FUNCTION_BLOCK FB_SetAxisMotion
VAR_IN_OUT
		axis : AXIS_REF;   			// the input axis
END_VAR
VAR_INPUT
	SetCmd : st_SetAxis;	
	ActStatus: st_ReadAxis;
END_VAR
VAR		
	fbMC_Stop:			MC_Stop;		
	fbMC_Home:			MC_Home;		
	fbMC_Halt:			MC_Halt;
	fbMC_Power:			MC_Power;
	fbMC_Reset:			MC_Reset;
	fbMC_MovVel:		MC_MoveVelocity;
	fbMC_MovAbs:		MC_MoveAbsolute;
	fbMC_MovConAbs:		MC_MoveContinuousAbsolute;//定义一个绝对运动功能块
	fbMC_MovRelative:	MC_MoveRelative;	

	eDir				:mc_direction;
	
	bWarning			:BOOL := FALSE;
	
	bHalt				:BOOL := FALSE;
	

END_VAR

CASE ActStatus.eState OF
	
	eAxis_ERRORSTOP:
		A_ErrorStop();	
	eAxis_DISABLED:
		A_Disable();	
	eAxis_STANDSTILL:
		A_Standstill();
	eAxis_HOMING:
		A_Homing();		
	eAxis_STOPPING:
		A_Stopping();	
	eAxis_DISCRETEMOTION:
		A_DiscreteMotion();		
	eAxis_CONTINOUSMOTION:
		A_ContinuousMotion();			
END_CASE
fbMC_Stop( Axis:= axis,Execute:= FALSE );
fbMC_Halt(Axis:=axis, Execute:= FALSE);
fbMC_Home( Axis:=axis, Execute:=FALSE);
fbMC_Reset(Axis:= axis, 	Execute:=FALSE);
fbMC_MovAbs(Axis:= axis, Execute:=FALSE);
fbMC_MovConAbs(Axis:= axis, Execute:=FALSE);
fbMC_MovRelative(Axis:= axis,  Execute:=FALSE);
fbMC_MovVel(Axis:= axis, Execute:=FALSE);

ACTION A_ContinuousMotion:
CASE SetCmd.eMC_Motion OF
	eMC_NONE:
		//fbMC_Halt(Axis:=axis, Execute:= TRUE);
	eMC_POWER:
		IF SetCmd.bEnable = TRUE THEN
			fbMC_Power(	Axis:= axis, Enable:= TRUE, Enable_Positive:= TRUE,
					Enable_Negative:= TRUE );
		ELSE
			fbMC_Power(	Axis:= axis, Enable:= FALSE);			
		END_IF	
		
	eMC_STOP:
		fbMC_Stop( Axis:= axis,Execute:= TRUE );
//		fbMC_Stop( Axis:= axis,Execute:= FALSE );
	
	eMC_HALT:
		fbMC_Halt(Axis:=axis, Execute:= TRUE);
//		fbMC_Halt(Axis:=axis, Execute:= FALSE);
		
	eMC_MOV_ABS:
		fbMC_MovAbs(Axis:= axis, Execute:=TRUE , 
					Position:=SetCmd.Position, 
					Velocity:=ABS(SetCmd.Velocity),
					BufferMode := MC_BlendingLow);
//		fbMC_MovAbs(Axis:= axis, Execute:=FALSE);
	
	eMC_MOV_CON_ABS:
		fbMC_MovConAbs(Axis:= axis, Execute:=TRUE, 
						Position:=SetCmd.Position ,Velocity:= ABS(SetCmd.Velocity),
						EndVelocity:= ABS(SetCmd.EndVelocity));
//		fbMC_MovConAbs(Axis:= axis, Execute:=FALSE);
	
	eMC_MOV_RELATIVE:
		fbMC_MovRelative(Axis:= axis,  Execute:=TRUE , 
			Distance:= SetCmd.Distance,  Velocity:= SetCmd.Velocity);
//		fbMC_MovRelative(Axis:= axis,  Execute:=FALSE);
	
	eMC_MOV_VEL:
		IF (SetCmd.Velocity >= 0) THEN
			eDir := MC_Positive_Direction;
		ELSE
			eDir := MC_Negative_Direction;
		END_IF
		fbMC_MovVel(Axis:= axis, Execute:=TRUE, 
					Velocity:=ABS(SetCmd.Velocity), Direction:=eDir);	
//		fbMC_MovVel(Axis:= axis, Execute:=FALSE);
		
ELSE
	bWarning := TRUE;
END_CASE
END_ACTION

ACTION A_Disable:
CASE SetCmd.eMC_Motion OF
	eMC_NONE:
	eMC_POWER:
		IF SetCmd.bEnable = TRUE THEN
			fbMC_Power(	Axis:= axis, Enable:= TRUE, Enable_Positive:= TRUE,
					Enable_Negative:= TRUE );
		ELSE
			fbMC_Power(	Axis:= axis, Enable:= FALSE);			
		END_IF
	eMC_Reset:
		fbMC_Reset(Axis:= axis, 	Execute:=TRUE);
//		fbMC_Reset(Axis:= axis, 	Execute:=FALSE);	
ELSE
	bWarning := TRUE;
END_CASE
END_ACTION

ACTION A_DiscreteMotion:
CASE SetCmd.eMC_Motion OF
	eMC_NONE:
		//fbMC_Halt(Axis:=axis, Execute:= TRUE);			
	eMC_POWER:
		IF SetCmd.bEnable = TRUE THEN
			fbMC_Power(	Axis:= axis, Enable:= TRUE, Enable_Positive:= TRUE,
					Enable_Negative:= TRUE );
		ELSE
			fbMC_Power(	Axis:= axis, Enable:= FALSE);			
		END_IF
	
	eMC_STOP:
		fbMC_Stop( Axis:= axis,Execute:= TRUE );
//		fbMC_Stop( Axis:= axis,Execute:= FALSE );
	
	eMC_HALT:
		fbMC_Halt(Axis:=axis, Execute:= TRUE);
//		fbMC_Halt(Axis:=axis, Execute:= FALSE);

	eMC_MOV_ABS:
		fbMC_MovAbs(Axis:= axis, Execute:=TRUE , 
					Position:=SetCmd.Position, 
					Velocity:=ABS(SetCmd.Velocity),
					BufferMode := MC_BlendingLow);
//		fbMC_MovAbs(Axis:= axis, Execute:=FALSE);
	
	eMC_MOV_CON_ABS:
		fbMC_MovConAbs(Axis:= axis, Execute:=TRUE, 
						Position:=SetCmd.Position ,Velocity:= ABS(SetCmd.Velocity),
						EndVelocity:= ABS(SetCmd.EndVelocity));
//		fbMC_MovConAbs(Axis:= axis, Execute:=FALSE);
	
	eMC_MOV_RELATIVE:
		fbMC_MovRelative(Axis:= axis,  Execute:=TRUE , 
			Distance:= SetCmd.Distance,  Velocity:= SetCmd.Velocity);
//		fbMC_MovRelative(Axis:= axis,  Execute:=FALSE);
	
	eMC_MOV_VEL:
		IF (SetCmd.Velocity >= 0) THEN
			eDir := MC_Positive_Direction;
		ELSE
			eDir := MC_Negative_Direction;
		END_IF
		fbMC_MovVel(Axis:= axis, Execute:=TRUE, 
					Velocity:=ABS(SetCmd.Velocity), Direction:=eDir);	
//		fbMC_MovVel(Axis:= axis, Execute:=FALSE);
		
ELSE
	bWarning := TRUE;
END_CASE
END_ACTION

ACTION A_ErrorStop:
CASE SetCmd.eMC_Motion OF
	eMC_NONE:
	eMC_RESET:	
		fbMC_Reset(Axis:= axis, 	Execute:=TRUE);		
//		fbMC_Reset(Axis:= axis, 	Execute:=FALSE);	
ELSE
	bWarning := TRUE;
END_CASE
END_ACTION

ACTION A_Homing:
CASE SetCmd.eMC_Motion OF
	eMC_NONE:	
	eMC_STOP:
		fbMC_Stop(Axis:=axis, 	Execute:=TRUE);
//		fbMC_Stop(Axis:=axis, 	Execute:=FALSE);
	eMC_POWER:
		IF SetCmd.bEnable = TRUE THEN
			fbMC_Power(	Axis:= axis, Enable:= TRUE, Enable_Positive:= TRUE,
					Enable_Negative:= TRUE );
		ELSE
			fbMC_Power(	Axis:= axis, Enable:= FALSE);			
		END_IF
ELSE
	bWarning := TRUE;		
END_CASE
END_ACTION

ACTION A_Standstill:
CASE SetCmd.eMC_Motion OF
	eMC_NONE:
	eMC_RESET:
		fbMC_Reset(Axis:= axis, 	Execute:=TRUE);

		bWarning := TRUE;	
	eMC_HOME:
		fbMC_Home( Axis:=axis, Execute:=TRUE ,
				   Position:=0 ,HomingMode:= );

	
	eMC_POWER:
		IF SetCmd.bEnable = TRUE THEN
			fbMC_Power(	Axis:= axis, Enable:= TRUE, Enable_Positive:= TRUE,
					Enable_Negative:= TRUE );
		ELSE
			fbMC_Power(	Axis:= axis, Enable:= FALSE);			
		END_IF	
		
	eMC_STOP:
		fbMC_Stop( Axis:= axis,Execute:= TRUE );

	
	eMC_HALT:
		fbMC_Halt(Axis:=axis, Execute:= TRUE);


	eMC_MOV_ABS:

		fbMC_MovAbs(Axis:= axis, Execute:=TRUE , 
					Position:= SetCmd.Position, 
					Velocity:= ABS(SetCmd.Velocity));

	
	eMC_MOV_CON_ABS:
		fbMC_MovConAbs(Axis:= axis, Execute:=TRUE, 
						Position:= SetCmd.Position ,Velocity:= ABS(SetCmd.Velocity),
						EndVelocity:= ABS(SetCmd.EndVelocity));

	
	eMC_MOV_RELATIVE:
		fbMC_MovRelative(Axis:= axis,  Execute:=TRUE , 
			Distance:= SetCmd.Distance,  Velocity:= ABS(SetCmd.Velocity));

	
	eMC_MOV_VEL:
		IF (SetCmd.Velocity >= 0) THEN
			eDir := MC_Positive_Direction;
		ELSE
			eDir := MC_Negative_Direction;
		END_IF
		fbMC_MovVel(Axis:= axis, Execute:=TRUE, 
					Velocity:=ABS(SetCmd.Velocity), Direction:=eDir);

ELSE
	bWarning := TRUE;	
END_CASE
END_ACTION

ACTION A_Stopping:
CASE SetCmd.eMC_Motion OF
	eMC_NONE:
	eMC_STOP:
		fbMC_Stop( Axis:= axis,Execute:= TRUE );
//		fbMC_Stop( Axis:= axis,Execute:= FALSE );		
	eMC_POWER:
		IF SetCmd.bEnable = TRUE THEN
			fbMC_Power(	Axis:= axis, Enable:= TRUE, Enable_Positive:= TRUE,
					Enable_Negative:= TRUE );
		ELSE
			fbMC_Power(	Axis:= axis, Enable:= FALSE);			
		END_IF
	
ELSE
	bWarning := TRUE;
END_CASE
END_ACTION

END_FUNCTION_BLOCK

(* stored: Version 1.1.0.1, ProductVersion 3.1.4022.12
   POU FB_SetAxisMotion: Id {3525fe16-db4c-4df2-b32e-c0850fa112d0}, SpecialFunc None
   Action A_ContinuousMotion: Id {a04b305e-d514-4023-9aee-01b7d802daa2}
   Action A_Disable: Id {e21ecd9d-08d6-4342-84ad-181e26702c9b}
   Action A_DiscreteMotion: Id {95b09518-3e6b-49c9-9f15-c1e96552aed8}
   Action A_ErrorStop: Id {047bd619-78a6-4151-b47f-544f83a81ae5}
   Action A_Homing: Id {3fc141f7-2cfe-4d25-a4e7-d1d0cc141eba}
   Action A_Standstill: Id {464e950c-3029-4c8e-adfc-23e09d0d37bd}
   Action A_Stopping: Id {13fbaf66-a053-4cc7-a61f-94880b765ed0} *)
